// TIA Portal project "test_24Vfischer_V2" (V17)

(* hardware
DEVICE "S7-1200-Station_1"  S7-1200 Station
   slot 0: "Baugruppenträger_0"  S7-1200 Rack  Rack  V1.0
   slot 1: "PLC_1"  CPU 1214C AC/DC/Rly  6ES7 214-1BG40-0XB0  V4.0
   slot 3: "AQ 1x12BIT_1"  AQ1 signal board  6ES7 232-4HA30-0XB0  V1.0
*)

// ===== PLC "PLC_1"  CPU 1214C AC/DC/Rly =====

VAR_GLOBAL   // PLC tag table "Standard-Variablentabelle"
   "-M1.rechts" AT %Q0.0 : Bool;   // drehen
   "-M1.links" AT %Q0.1 : Bool;
   "-M2.rechts" AT %Q0.2 : Bool;   // hoch
   "-M2.links" AT %Q0.3 : Bool;   // runter
   "-M3.rechts" AT %Q0.4 : Bool;   // vor
   "-M3.links" AT %Q0.5 : Bool;   // zurück
   "-M4.rechts" AT %Q0.6 : Bool;   // auf
   "-M4.links" AT %Q0.7 : Bool;   // zu
   "-I1" AT %I0.0 : Bool;   // Enc drehen
   "-I2" AT %I0.1 : Bool;   // Enc hoch runter
   "-I3" AT %I0.2 : Bool;   // Enc vor zurück
   "-I4" AT %I0.3 : Bool;   // Enc auf zu
   "-I5" AT %I0.4 : Bool;   // Endl drehen
   "-I6" AT %I0.5 : Bool;   // Endl hoch runter
   "-I7" AT %I0.6 : Bool;   // Endl vor zurück
   "-I8" AT %I0.7 : Bool;   // Endl auf zu
END_VAR

DATA_BLOCK "Baustein_1_DB"   // DB1
{ S7_Optimized_Access := 'TRUE' }
VERSION : 0.1
// stored: InstanceOfName Baustein_1
"Baustein_1"
BEGIN
END_DATA_BLOCK

DATA_BLOCK "Ausgänge_DB"   // DB2
{ S7_Optimized_Access := 'TRUE' }
VERSION : 0.1
// stored: InstanceOfName Ausgänge
"Ausgänge"
BEGIN
END_DATA_BLOCK

FUNCTION_BLOCK "Baustein_1"   // FB1, FBD
{ S7_Optimized_Access := 'TRUE' }
VERSION : 0.1
   VAR_INPUT
      "Enc drehen" : Bool;
      "Enc hoch runter" : Bool;
      "Enc vor zurück" : Bool;
      "Enc auf zu" : Bool;
      "Endl hoch runter" : Bool;
      "Endl drehen" : Bool;
      "Endl vor zurück" : Bool;
      "Endl auf zu" : Bool;
   END_VAR
   VAR_OUTPUT
      hoch : Bool;
      runter : Bool;
      "rechts drehen" : Bool;
      "links drehen" : Bool;
      vor : Bool;
      zurück : Bool;
      auf : Bool;
      zu : Bool;
      hoch1 : Bool;
      hoch2 : Bool;
      runter1 : Bool;
      runter2 : Bool;
      rechts1 : Bool;
      rechts2 : Bool;
      links1 : Bool;
      links2 : Bool;
      vor1 : Bool;
      vor2 : Bool;
      zurück1 : Bool;
      zurück2 : Bool;
      auf1 : Bool;
      auf2 : Bool;
      zu1 : Bool;
      zu2 : Bool;
   END_VAR
   VAR RETAIN
      IEC_Counter_0_Instance : CTUD_INT;
      IEC_Counter_0_Instance_1 : CTU_INT;
   END_VAR
   VAR
      Schritt1 : Bool;
      Schritt2 : Bool;
      Schritt3 : Bool;
      Schritt4 : Bool;
      Schritt5 : Bool;
      Initialschritt : Bool;
      Schritt6 : Bool;
      "Schritt 7" : Bool;
      Schritt8 : Bool;
      Schritt9 : Bool;
      Schritt10 : Bool;
      Schritt11 : Bool;
      Schritt12 : Bool;
      initialisieren : Bool;
      test : Bool;
      "Zähler vor zurück" : Int;
      "vor ende" : Bool;
      "zu ende" : Bool;
   END_VAR
   VAR RETAIN
      IEC_Counter_0_Instance_2 : CTU_INT;
      IEC_Counter_0_Instance_3 : CTU_INT;
   END_VAR
   VAR
      IEC_Timer_0_Instance : TON_TIME;
      IEC_Timer_0_Instance_1 : TON_TIME;
   END_VAR
   VAR RETAIN
      IEC_Counter_0_Instance_4 : CTU_INT;
   END_VAR
   VAR
      IEC_Timer_0_Instance_2 : TON_TIME;
      IEC_Timer_0_Instance_3 : TON_TIME;
   END_VAR
BEGIN

REGION Network 2
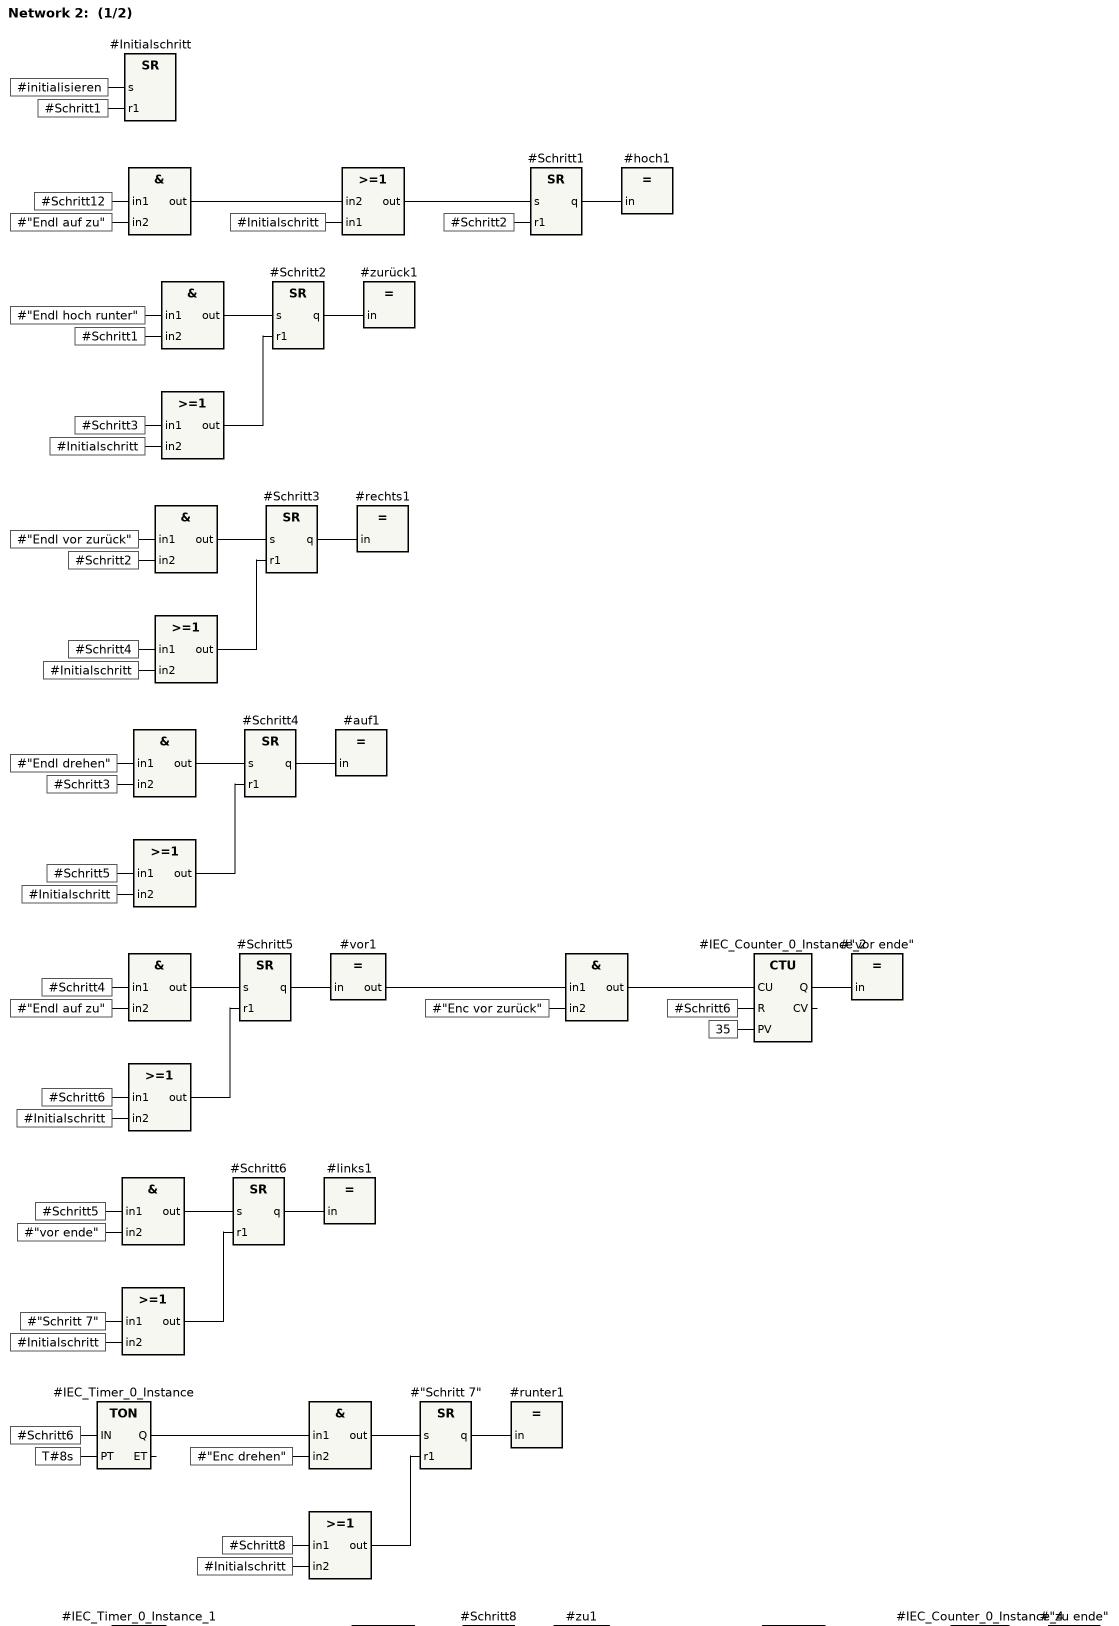
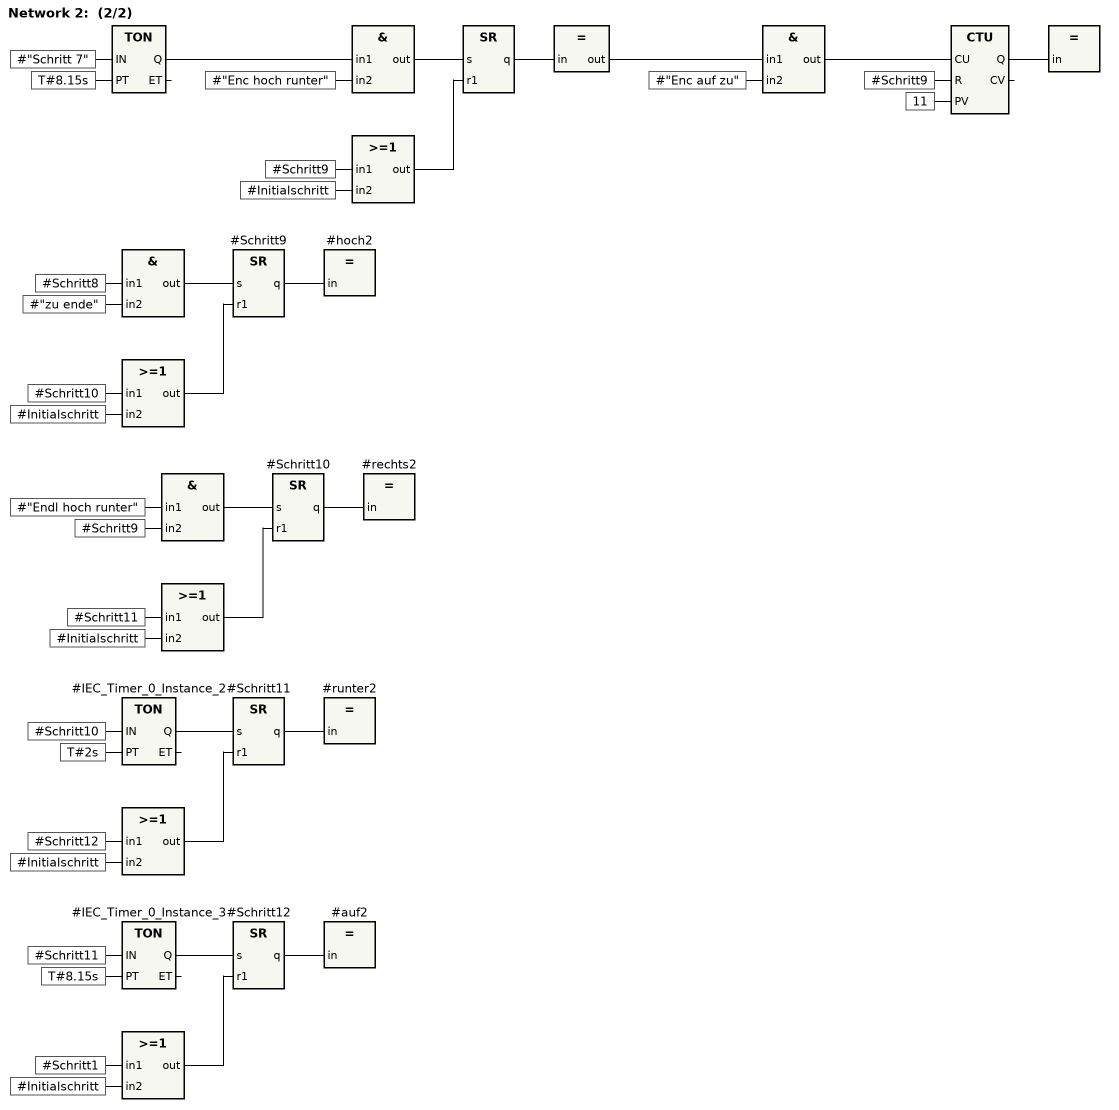
   IF #initialisieren THEN
       #Initialschritt := TRUE;   // SR flip-flop
   END_IF;
   IF #Schritt1 THEN #Initialschritt := FALSE; END_IF;
   IF (#Schritt12 AND #"Endl auf zu") OR #Initialschritt THEN
       #Schritt1 := TRUE;   // SR flip-flop
   END_IF;
   IF #Schritt2 THEN #Schritt1 := FALSE; END_IF;
   #hoch1 := #Schritt1;
   IF #"Endl hoch runter" AND #Schritt1 THEN
       #Schritt2 := TRUE;   // SR flip-flop
   END_IF;
   IF #Schritt3 OR #Initialschritt THEN #Schritt2 := FALSE; END_IF;
   #zurück1 := #Schritt2;
   IF #"Endl vor zurück" AND #Schritt2 THEN
       #Schritt3 := TRUE;   // SR flip-flop
   END_IF;
   IF #Schritt4 OR #Initialschritt THEN #Schritt3 := FALSE; END_IF;
   #rechts1 := #Schritt3;
   IF #"Endl drehen" AND #Schritt3 THEN
       #Schritt4 := TRUE;   // SR flip-flop
   END_IF;
   IF #Schritt5 OR #Initialschritt THEN #Schritt4 := FALSE; END_IF;
   #auf1 := #Schritt4;
   IF #Schritt4 AND #"Endl auf zu" THEN
       #Schritt5 := TRUE;   // SR flip-flop
   END_IF;
   IF #Schritt6 OR #Initialschritt THEN #Schritt5 := FALSE; END_IF;
   #vor1 := #Schritt5;
   #IEC_Counter_0_Instance_2(CU := #Schritt5 AND #"Enc vor zurück", R := #Schritt6, PV := 35);   // CTU
   #"vor ende" := #IEC_Counter_0_Instance_2.Q;
   IF #Schritt5 AND #"vor ende" THEN
       #Schritt6 := TRUE;   // SR flip-flop
   END_IF;
   IF #"Schritt 7" OR #Initialschritt THEN #Schritt6 := FALSE; END_IF;
   #links1 := #Schritt6;
   #IEC_Timer_0_Instance(IN := #Schritt6, PT := T#8s);   // TON
   IF #IEC_Timer_0_Instance.Q AND #"Enc drehen" THEN
       #"Schritt 7" := TRUE;   // SR flip-flop
   END_IF;
   IF #Schritt8 OR #Initialschritt THEN #"Schritt 7" := FALSE; END_IF;
   #runter1 := #"Schritt 7";
   #IEC_Timer_0_Instance_1(IN := #"Schritt 7", PT := T#8.15s);   // TON
   IF #IEC_Timer_0_Instance_1.Q AND #"Enc hoch runter" THEN
       #Schritt8 := TRUE;   // SR flip-flop
   END_IF;
   IF #Schritt9 OR #Initialschritt THEN #Schritt8 := FALSE; END_IF;
   #zu1 := #Schritt8;
   #IEC_Counter_0_Instance_4(CU := #Schritt8 AND #"Enc auf zu", R := #Schritt9, PV := 11);   // CTU
   #"zu ende" := #IEC_Counter_0_Instance_4.Q;
   IF #Schritt8 AND #"zu ende" THEN
       #Schritt9 := TRUE;   // SR flip-flop
   END_IF;
   IF #Schritt10 OR #Initialschritt THEN #Schritt9 := FALSE; END_IF;
   #hoch2 := #Schritt9;
   IF #"Endl hoch runter" AND #Schritt9 THEN
       #Schritt10 := TRUE;   // SR flip-flop
   END_IF;
   IF #Schritt11 OR #Initialschritt THEN #Schritt10 := FALSE; END_IF;
   #rechts2 := #Schritt10;
   #IEC_Timer_0_Instance_2(IN := #Schritt10, PT := T#2s);   // TON
   IF #IEC_Timer_0_Instance_2.Q THEN
       #Schritt11 := TRUE;   // SR flip-flop
   END_IF;
   IF #Schritt12 OR #Initialschritt THEN #Schritt11 := FALSE; END_IF;
   #runter2 := #Schritt11;
   #IEC_Timer_0_Instance_3(IN := #Schritt11, PT := T#8.15s);   // TON
   IF #IEC_Timer_0_Instance_3.Q THEN
       #Schritt12 := TRUE;   // SR flip-flop
   END_IF;
   IF #Schritt1 OR #Initialschritt THEN #Schritt12 := FALSE; END_IF;
   #auf2 := #Schritt12;
END_REGION
END_FUNCTION_BLOCK

FUNCTION_BLOCK "Ausgänge"   // FB2, FBD
{ S7_Optimized_Access := 'TRUE' }
VERSION : 0.1
BEGIN

REGION Network 1
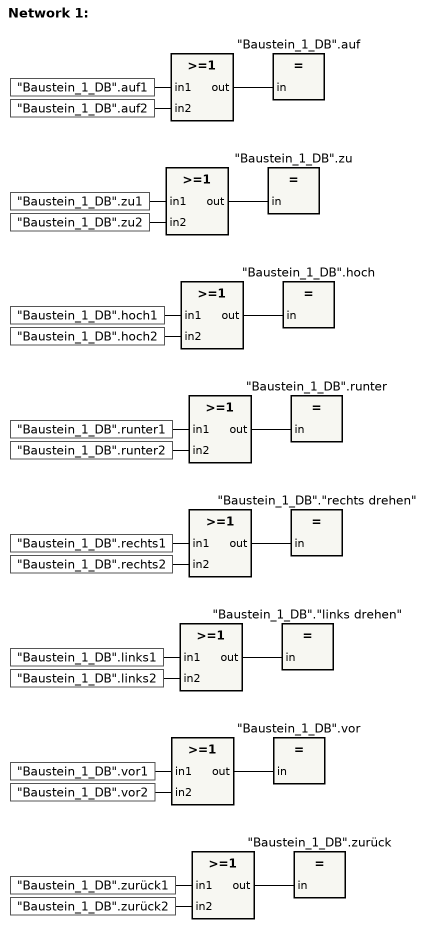
   "Baustein_1_DB".auf := "Baustein_1_DB".auf1 OR "Baustein_1_DB".auf2;
   "Baustein_1_DB".zu := "Baustein_1_DB".zu1 OR "Baustein_1_DB".zu2;
   "Baustein_1_DB".hoch := "Baustein_1_DB".hoch1 OR "Baustein_1_DB".hoch2;
   "Baustein_1_DB".runter := "Baustein_1_DB".runter1 OR "Baustein_1_DB".runter2;
   "Baustein_1_DB"."rechts drehen" := "Baustein_1_DB".rechts1 OR "Baustein_1_DB".rechts2;
   "Baustein_1_DB"."links drehen" := "Baustein_1_DB".links1 OR "Baustein_1_DB".links2;
   "Baustein_1_DB".vor := "Baustein_1_DB".vor1 OR "Baustein_1_DB".vor2;
   "Baustein_1_DB".zurück := "Baustein_1_DB".zurück1 OR "Baustein_1_DB".zurück2;
END_REGION
END_FUNCTION_BLOCK

ORGANIZATION_BLOCK "Main"   // OB1, FBD, ProgramCycle
TITLE = "Main Program Sweep (Cycle)"
{ S7_Optimized_Access := 'TRUE' }
VERSION : 0.1
   VAR_INPUT
      Initial_Call : Bool;   // Initial call of this OB
      Remanence : Bool;   // =True, if remanent data are available
   END_VAR
BEGIN

REGION Network 1
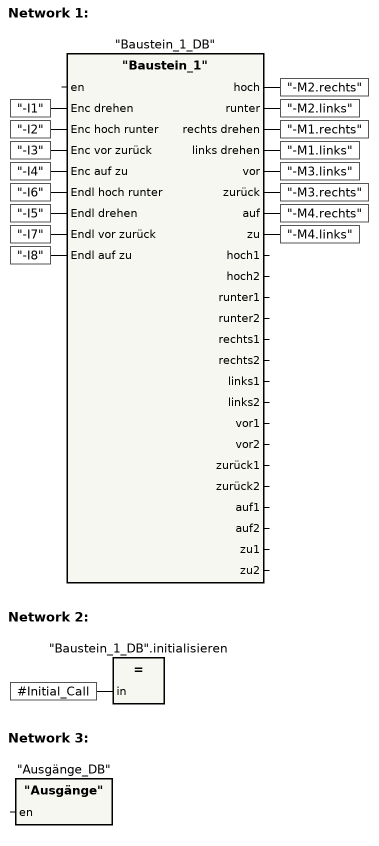
   "Baustein_1_DB"("Enc drehen" := "-I1",   // "Baustein_1"
                   "Enc hoch runter" := "-I2",
                   "Enc vor zurück" := "-I3",
                   "Enc auf zu" := "-I4",
                   "Endl hoch runter" := "-I6",
                   "Endl drehen" := "-I5",
                   "Endl vor zurück" := "-I7",
                   "Endl auf zu" := "-I8",
                   hoch => "-M2.rechts",
                   runter => "-M2.links",
                   "rechts drehen" => "-M1.rechts",
                   "links drehen" => "-M1.links",
                   vor => "-M3.links",
                   zurück => "-M3.rechts",
                   auf => "-M4.rechts",
                   zu => "-M4.links");
END_REGION

REGION Network 2
   "Baustein_1_DB".initialisieren := #Initial_Call;
END_REGION

REGION Network 3
   "Ausgänge_DB"();   // "Ausgänge"
END_REGION
END_ORGANIZATION_BLOCK